FUNCTION_BLOCK RQST_GEN (* FBMGT Request Generator *)
  (* Standard: 61499 ITA; ApplicationDomain: Device Management; Function: FBMGT Request Generator *)
  (* Version 0.1, 2007-11-08, JHC, Holobloc Inc, Changed RQST to OUT; subclassed from FBFunction. *)
  (* Version 0.0, 2001-11-27, JHC, Rockwell Automation, Copied/modified from QUERY_GEN. *)
  (* Compiler header: package fb.rt.ita; import fb.rt.math.FBFunction; *)
  (* Compiler classdef: public class RQST_GEN extends FBFunction *)
  (* Compiler Java Sun JDK 1.6.0 *)
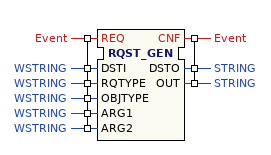
  EVENT_INPUT
    REQ WITH DSTI, RQTYPE, OBJTYPE, ARG1, ARG2;
  END_EVENT
  EVENT_OUTPUT
    CNF WITH DSTO, OUT;
  END_EVENT
  VAR_INPUT
    DSTI : WSTRING; (* Destination *)
    RQTYPE : WSTRING; (* CREATE,DELETE,READ,WRITE,QUERY *)
    OBJTYPE : WSTRING; (* FB,Connection *)
    ARG1 : WSTRING; (* FB Name or Connection Source *)
    ARG2 : WSTRING; (* FB Type or Connection Destination *)
  END_VAR
  VAR_OUTPUT
    DSTO : STRING; (* DSTI converted to STRING *)
    OUT : STRING; (* FBMGT request *)
  END_VAR
END_FUNCTION_BLOCK
